FUNCTION_BLOCK AE_DELAY (* Delayed event propagation (AE Adapter) *)
  (* Standard: 61499-2; Description: Copyright (c) 2026 HR Agrartechnik GmbH This program and the accompanying materials are made available under the terms of the Eclipse Public License 2.0 which is available at https://www.eclipse.org/legal/epl-2.0/ SPDX-License-Identifier: EPL-2.0 *)
  (* Version 1.0, 2026-02-01, Franz Höpfinger, HR Agrartechnik GmbH, Wrapper for E_DELAY using AE adapters *)
  PACKAGE adapter::events::unidirectional::timers;
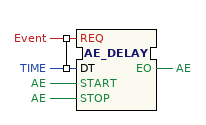
  EVENT_INPUT
    REQ WITH DT; (* Update DT *)
  END_EVENT
  VAR_INPUT
    DT : TIME; (* Delay time *)
  END_VAR
  SOCKETS
    START : adapter::types::unidirectional::AE; (* Start delay *)
    STOP : adapter::types::unidirectional::AE; (* Stop delay *)
  END_SOCKETS
  PLUGS
    EO : adapter::types::unidirectional::AE; (* Delayed event *)
  END_PLUGS
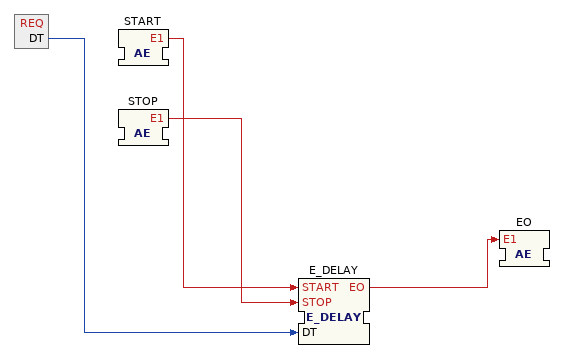
  FBS
    E_DELAY : iec61499::events::E_DELAY;
  END_FBS
  EVENT_CONNECTIONS
    START.E1 TO E_DELAY.START;
    STOP.E1 TO E_DELAY.STOP;
    E_DELAY.EO TO EO.E1;
  END_CONNECTIONS
  DATA_CONNECTIONS
    DT TO E_DELAY.DT;
  END_CONNECTIONS
END_FUNCTION_BLOCK
